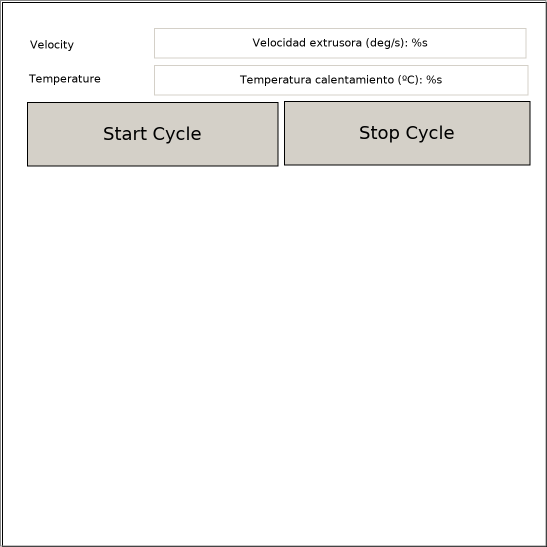
VISUALIZATION BasicHMI  // 547x547
    Rectangle (2,2 545x545)
    Textfield (154,28 372x30), "Velocidad extrusora (deg/s): %s", text variable: HMI.Tb_Vel
        OnMouseDown: write HMI.Tb_Vel via VisuDialogs.Numpad
    Label (27,30 120x30), "Velocity"
    Rectangle (27,102 251x64), "Start Cycle"
        tap HMI.Bt_StartCycle
    Label (26,64 120x30), "Temperature"
    Textfield (154,65 374x30), "Temperatura calentamiento (ºC): %s", text variable: HMI.Tb_Temp
        OnMouseDown: write HMI.Tb_Temp via VisuDialogs.Keypad
    Rectangle (284,101 246x64), "Stop Cycle"
        tap HMI.Bt_StopCycle
END_VISUALIZATION

(* stored: Version 1.1.0.1, ProductVersion 3.1.4024.9
   Visu BasicHMI: Id {8b998f78-e1f7-4f21-9e56-fbd1f3cc78cf} *)
